(* This function block implements basic functionality for Isolation Gate Valves*)
(* This function block interlock is as follows:
1. The valve can be opened when the difference between the pressures on both sides is
less than the maximum differential pressure.
2. This rule persists until the pressures on both sides are lower than the vacuum-setpoint.
3. Once at-vac, the valve will close if the pressure on either side rises above the setpoint.*)
(*This function block also implements PMPS and EPS interlocks, as well as Fast MPS trigger*)
{attribute 'no_check'}
{attribute 'reflection'} 
FUNCTION_BLOCK FB_VGC_tst Extends FB_Valve
VAR_IN_OUT
	
END_VAR
VAR_INPUT
	(*Upstream Gauge, usually ion gauge*)
	i_stUSG	:	ST_VG;
	(*Downstream Gauge, usually ion gauge*)
	i_stDSG	:	ST_VG;
	{attribute 'pytmc' := '
    pv: Dis_DPIlk
	'}
	i_xDis_DPIlk : BOOL := FALSE;  (* Set to true when calling the function to disable the differential pressure interlock *)
	i_xPMPS_OK:	BOOL	; (*Set to True To switch of the bptm*)
	{attribute 'pytmc' := '
    pv: EPS_OK
	'}
	i_xEPS_OK:	BOOL	:= TRUE; (*External EPS interlock, Set to TRUE when no EPS interlock is required, otherwise set to correct interlock signal*)
	i_xExt_OK: BOOL; (*Other External Interlock, Set to True when no external interlock is required. If this Valve is neigboring a Fast Shutter this should be linked to the fast shutter xVAC_FAULT_OK*)
	i_xOverrideMode : BOOL; (*To be linked to global override bit. This Overrides Vacuum logic only, EPS, MPS and PMPS are still enforces*)
	// Reset fault
	{attribute 'pytmc' := '
    pv: FF_Reset
	'}
    i_xReset: BOOL;
	i_xIsAperture:BOOL :=FALSE; // Set tp True if this is an Aperture Valve, the MPS Fault will trip only when moving.
	i_sDevName : T_MaxString :=  'VGC'; // Device name for diagnostic
	i_nTransitionRootID: UDINT; //A unique transition Root ID that is equal to or greater than 1000
END_VAR
VAR_OUTPUT
	{attribute 'pytmc' := '
    pv:
	'}
	iq_stValve : ST_VGC; (* All valve data and states will be in this struct*)
	
	{attribute 'pytmc' := '
    pv: MPS_FAULT_OK
	field: ZNAM MPS FAULT ;
	field: ONAM MPS OK ;
	'}
	xMPS_OK:	BOOL; (*MPS Fast OK, is set when the Valve is Open*)
END_VAR
VAR_IN_OUT
	io_fbFFHWO    :    FB_HardwareFFOutput;
	fbArbiter: FB_Arbiter();
END_VAR
VAR
	// PMPS
	{attribute 'pytmc' := '
    pv: MPS_OK
	'}
	xPMPS_OK:	BOOL	; (*PMPS interlock*)
	bMoving : BOOL;
	bDone :BOOL;
	tBPTMtimeout:TON;
	 i_nRequestedAssertionID:DWORD;
	bptm: BeamParameterTransitionManager;  
	FFO    :    FB_FastFault :=(
        i_DevName := 'VGC',
        i_Desc := 'Fault occurs when the valve is not in open state',
        i_TypeCode := 16#1010);
	//g_FastFaultOutput1	:	FB_HardwareFFOutput;	

	{attribute 'instance-path'}
	{attribute 'noinit'}
	sPath: STRING;
	
	rDiffPressAllowed	:	REAL := 22.5; // Torr, Default value comes from Vat Valve Manual
	rDiffPress : REAL;
	set : BOOL;
    reset: BOOL;
	  
	xFirstPass	:	BOOL;
	fbFSInit		:	R_TRIG;
	
	tonDelOK : TON;
	rtOK	:	R_TRIG;
	tonOvrd	:	TON;
	rtOpen	:	R_TRIG;
	ftClose: F_TRIG;
	
	tDelOK	:	TIME := T#60S;
	tOvrd	:	TIME := T#10s;
	
	
	(* Timeouts*)
	tTimeOutDuration: TIME:= T#30S;
	tOPNtimeout: TON;
	tCLStimeout:TON;
	
	
	(*IO*)
	i_xOpnLS	AT%I*: BOOL;
	i_xClsLS	AT%I*: BOOL;
	q_xOPN_DO	AT%Q*: BOOL;
    
    // For logging
    eVGCPrevState : E_VGC;
 
	
END_VAR

(* Vacuum gate valve
A. Wallace
16-10-29

A gate valve isolates vacuum volumes. Ideally it can be opened when a system is vented
to allow for faster pumping, and will close when high vacuum is lost.

The following behavior is good for valves in something like a gas attenuator.
This function block does the following:
1. The valve can be opened when the difference between the pressures on both sides is
less than the maximum differential pressure.
2. This rule persists until the pressures on both sides are lower than the vacuum-setpoint.
3. Once at-vac, the valve will close if the pressure on either side rises above the setpoint.

Alternatively, the differential pressure interlock can be disabled so the valve may only be opened
if the pressure on both sides is lower than the at-vacuum-setpoint. You want this behavior if 
the valve is to be used in a UHV section.

Hysteresis is employed to ensure a smooth transition from vented/pumping down, to at-vac.

Finally, an override system is built in so you can bypass all the interlocking logic and 
get back online.
*)
(* 10/1/2018 Margaret Ghaly included EPS, PMPS Checkes and MPS trigger signals*)


fbFSInit( CLK := TRUE, Q => xFirstPass);
(*IO Mapping*)
ACT_IO();

(* On first PLC pass, put valve into vented state, which implies a closed valve *)
IF xFirstPass THEN
	iq_stValve.eVGC_State := Vented;
	iq_stValve.pv_xOPN_SW := FALSE;
	FFO.i_DevName := i_sDevName;
END_IF


///Check valve position
IF iq_stValve.i_xClsLS AND  iq_stValve.i_xOpnLS THEN
	iq_stValve.eState:=INVALID;
ELSIF NOT iq_stValve.i_xClsLS AND iq_stValve.i_xOpnLS AND iq_stValve.q_xOPN_DO THEN 
	iq_stValve.eState:=OPEN;
ELSIF NOT iq_stValve.i_xClsLS AND iq_stValve.i_xOpnLS AND NOT iq_stValve.q_xOPN_DO THEN 
	iq_stValve.eState:=OPEN_F;
ELSIF iq_stValve.i_xClsLS AND NOT iq_stValve.i_xOpnLS AND NOT iq_stValve.q_xOPN_DO THEN 
	iq_stValve.eState:=CLOSED;
ELSIF NOT iq_stValve.i_xClsLS AND NOT iq_stValve.i_xOpnLS THEN 
	iq_stValve.eState:=MOVING;
ELSE
	iq_stValve.eState:=INVALID;
END_IF

// Update hysteresis
///////////////////////////////////////////////////
IF iq_stValve.rAT_VAC_SP_LAST <> iq_stValve.rAT_VAC_SP OR xFirstPass THEN
	iq_stValve.rAT_VAC_SP_LAST := iq_stValve.rAT_VAC_SP;
	iq_stValve.rAT_VAC_HYS := iq_stValve.rHYST_PERC * iq_stValve.rAT_VAC_SP;
END_IF

iq_stValve.rAT_VAC_HYS := LIMIT(0, iq_stValve.rAT_VAC_HYS, iq_stValve.rAT_VAC_SP);
IF iq_stValve.rAT_VAC_SP <> 0 THEN
	IF iq_stValve.rHYST_PERC <> (iq_stValve.rAT_VAC_HYS / iq_stValve.rAT_VAC_SP) THEN
		iq_stValve.rHYST_PERC := LIMIT(0, (iq_stValve.rAT_VAC_HYS / iq_stValve.rAT_VAC_SP) ,1);
	END_IF
END_IF
// Valve at vacuum check
///////////////////////////////////////////////////
	set := i_stUSG.rPRESS < iq_stValve.rAT_VAC_HYS AND i_stDSG.rPRESS < iq_stValve.rAT_VAC_HYS AND i_stUSG.xPRESS_OK AND i_stDSG.xPRESS_OK;
 	iq_stValve.xAT_VAC S= set;
	reset := i_stUSG.rPRESS > iq_stValve.rAT_VAC_SP OR i_stDSG.rPRESS > iq_stValve.rAT_VAC_SP OR NOT i_stUSG.xPRESS_OK OR NOT i_stDSG.xPRESS_OK;
	iq_stValve.xAT_VAC R= reset;
	
// Differential pressure check
///////////////////////////////////////////////////
	(* Calc the differential pressure across the valve *)
	rDiffPress := ABS(i_stUSG.rPRESS - i_stDSG.rPRESS);
	
	(* As long as the differential pressure is less than 30mbar, the valve is allowed to open *)
	IF rDiffPress <= rDiffPressAllowed AND i_stUSG.xPRESS_OK AND i_stDSG.xPRESS_OK THEN
		iq_stValve.xDP_OK := TRUE;
	ELSE
		iq_stValve.xDP_OK	:= FALSE;
		(* If the differential pressure is exceeded, even when the valve is open,
		the state is unexpected and triggers a fault, because it suggests that something
		is wrong with the valve, or gauges or mapping or there is a major leak on one side.*)
		iq_stValve.eVGC_State := ERR_DiffPress;
        iq_stValve.xERR_DifPres := TRUE;
	END_IF

// Valve state
///////////////////////////////////////////////////
CASE iq_stValve.eVGC_State OF
	Vented: (* The Vented state is used during pump down *)        
		(* Assuming the pump down went well, we are now at vacuum on both sides,
		so we move to the vacuum state, otherwise remain in the vented state *)
		IF iq_stValve.xAT_VAC AND (NOT (iq_stValve.xERR_DifPres)) AND (NOT (iq_stValve.xERR_SP)) AND (NOT (iq_stValve.xERR_ExtFault))THEN
		    iq_stValve.eVGC_State := AtVacuum;
		ELSE
		    iq_stValve.eVGC_State := Vented;
		END_IF
	
	AtVacuum:
		IF iq_stValve.xAT_VAC THEN
		(* If both pressure setpoints are made,
		then enable the differential pressure interlock, regardless of the valve state
		assuming we're using some kind of ion gauge where a pressure setpoint cannot be higher than 1E-4 T *)
		iq_stValve.eVGC_State := AtVacuum;
				
		ELSE
		
			(* If the valve is open (or in an unknown state) and either gauge is not at it's vacuum setpoint,
			we have a loss of vacuum error *)
			IF (iq_stValve.i_xOpnLS OR (NOT iq_stValve.i_xOpnLS AND NOT iq_stValve.i_xClsLS)) THEN
				iq_stValve.eVGC_State := ERR_LostVac;
				iq_stValve.xERR_SP := TRUE; //TAW changed this to the ERR_SP bool because I think that's what it was intended to be?
		
			(* Alternatively, if the valve is already closed and we lose pressure on one side,
			it was probably intentional venting, so we calmly move back to venting mode, and
			disable the differential pressure interlock *) //?? 
			ELSIF iq_stValve.i_xClsLS THEN
				iq_stValve.eVGC_State := Vented;
			END_IF
		
		END_IF
	
	ERR_DiffPress:       
		IF NOT (iq_stValve.xERR_DifPres) THEN
			IF iq_stValve.xAT_VAC AND (NOT (iq_stValve.xERR_DifPres)) AND (NOT (iq_stValve.xERR_SP)) AND (NOT (iq_stValve.xERR_ExtFault))THEN
		    	iq_stValve.eVGC_State := AtVacuum;
			ELSE
		    	iq_stValve.eVGC_State := Vented;
			END_IF
		END_IF
		
	
	ERR_LostVac:
		IF NOT (iq_stValve.xERR_SP) THEN
			IF iq_stValve.xAT_VAC AND (NOT (iq_stValve.xERR_DifPres)) AND (NOT (iq_stValve.xERR_SP)) AND (NOT (iq_stValve.xERR_ExtFault))THEN
		    	iq_stValve.eVGC_State := AtVacuum;
			ELSE
		    	iq_stValve.eVGC_State := Vented;
			END_IF
		END_IF
		
	ERR_ExtFault:
		IF NOT (iq_stValve.xERR_ExtFault) AND (i_xExt_OK) THEN
			IF iq_stValve.xAT_VAC AND (NOT (iq_stValve.xERR_DifPres)) AND (NOT (iq_stValve.xERR_SP)) AND (NOT (iq_stValve.xERR_ExtFault))THEN
		    	iq_stValve.eVGC_State := AtVacuum;
			ELSE
		    	iq_stValve.eVGC_State := Vented;
			END_IF
		END_IF
END_CASE

IF (NOT i_xExt_OK) AND (iq_stValve.eState=OPEN)  THEN
	iq_stValve.eVGC_State := ERR_ExtFault;
	iq_stValve.xERR_ExtFault := TRUE;
END_IF

// Interlock evaluation - with bypass for DP ILK bypass
///////////////////////////////////////////////
IF i_xDis_DPIlk THEN
	iq_stValve.xOPN_OK := iq_stValve.xEXT_OK; // AND iq_stValve.xDP_OK ;
ELSE
	iq_stValve.xOPN_OK := iq_stValve.xEXT_OK AND iq_stValve.xAT_VAC;
END_IF


(* Valve operation *)

(* Override logic *)
(* Goal: give ability to override, but do so in a way that people won't forget it.
Solution: Override only after ten seconds of override, protect against blips,
when the valve permission goes true for more than ten seconds consistently, remove override
*)

tonDelOK(IN:=iq_stValve.xOPN_OK, PT:=tDelOK);
rtOK(CLK:=tonDelOK.Q);
IF rtOK.Q AND iq_stValve.pv_xOvrdOpn THEN 
	iq_stValve.pv_xOvrdOpn :=FALSE;
	if (iq_stValve.eState = OPEN) AND (i_xOverrideMode) THEN iq_stValve.pv_xOPN_SW := TRUE; END_IF //for seamless transition   
    //Log
    fbLogger(sMsg:='Override expired', eSevr:=TcEventSeverity.Warning);
END_IF
// Release the Force Open bit when the system override is false
IF NOT (i_xOverrideMode) THEN  iq_stValve.pv_xOvrdOpn :=FALSE; END_IF
//Override timer
tonOvrd(IN:=iq_stValve.pv_xOvrdOpn, PT:=tOvrd);


(* Valve operation *)
(* Here's where we evaluate sw actions and operate the valve *)
(* Valve operation *)

ftClose(CLK:= iq_stValve.pv_xOPN_SW);
rtOpen(CLK:= iq_stValve.pv_xOPN_SW);

(*PMPS OPERATION AND BPTM*)
(*PMPS*)
IF NOT(i_xPMPS_OK) THEN
	ACT_PMPS();
END_IF
xPMPS_OK := i_xPMPS_OK OR (bptm.q_xTransitionAuthorized OR tBPTMtimeout.Q);
(*when interlock is lost the Valve closes regardless of the status of the PMPS and EPS*)
IF NOT (iq_stValve.xOPN_OK) THEN
	iq_stValve.pv_xOPN_SW:= FALSE; // Reset switch after inlk is lost
	iq_stValve.q_xOPN_DO := (iq_stValve.pv_xOPN_SW  AND iq_stValve.xOPN_OK) OR (tonOvrd.Q AND i_xOverrideMode);
ELSIF xPMPS_OK THEN 
	iq_stValve.q_xOPN_DO := (iq_stValve.pv_xOPN_SW  AND iq_stValve.xOPN_OK) OR (tonOvrd.Q AND i_xOverrideMode);
END_IF

(*MPS Fault setting*)
If (i_xIsAperture ) THEN 
	(* When the valve  is open or in Closed position MPS is OK, Fault while moving*)
	xMPS_OK := i_xOpnLS XOR i_xClsLS; 
ELSE
	(* When the valve  is open MPS is OK*)
	xMPS_OK := i_xOpnLS AND NOT i_xClsLS AND q_xOPN_DO; 
END_IF


///Check valve moving postion timout
IF NOT iq_stValve.i_xClsLS AND tCLStimeout.Q THEN 
	iq_stValve.bErrorPresent := TRUE;
	iq_stValve.sErrorMessage := 'Close Timeout';
ELSIF NOT iq_stValve.i_xOpnLS AND tOPNtimeout.Q THEN 
	iq_stValve.bErrorPresent := TRUE; 
	iq_stValve.sErrorMessage := 'Open Timeout';
END_IF
IF (iq_stValve.eState=INVALID) THEN
	iq_stValve.bErrorPresent := TRUE; 
	iq_stValve.sErrorMessage := CONCAT(sPath,'Invalid Valve Position');
END_IF


(*Timers*)
tOPNtimeout(IN:= iq_stValve.q_xOPN_DO, PT := tTimeOutDuration );
tCLStimeout(IN:= NOT iq_stValve.q_xOPN_DO, PT := tTimeOutDuration);


// Alarm reset
//////////////////////////////////////
ACT_ResetAlarms();

(*IO Mapping*)
ACT_IO();

// Log States and triggers
ACT_Logger();



(*FAST FAULT*)
FFO(i_xOK := xMPS_OK,
    i_xReset := i_xReset,
	i_xAutoReset :=TRUE,
    io_fbFFHWO := io_fbFFHWO);

ACTION ACT_IO:
(*inputs*)
iq_stValve.i_xOpnLS := 	i_xOpnLS;
iq_stValve.i_xClsLS:=	i_xClsLS;
iq_stValve.xEXT_OK := i_xEXT_OK;
iq_stValve.xOverrideMode := i_xOverrideMode;
(*outputs*)
q_xOPN_DO:= iq_stValve.q_xOPN_DO;

(*ILK Devices*)
iq_stValve.sIlkUSDeviceName := This^.i_stUSG.sPath;
iq_stValve.sIlkDSDeviceName := This^.i_stDSG.sPath;
END_ACTION

ACTION ACT_Logger:
// ILK logger

IF NOT (iq_stValve.xOPN_OK) AND (ePrevState = OPEN) AND NOT (TonOvrd.Q) THEN
 		fbLogger(sMsg:='Lost interlock ok bit while valve was open.', eSevr:=TcEventSeverity.Critical);  	
END_IF


//Positiong STATE Logger  
IF ePrevState <> iq_stValve.eState THEN
	  CASE iq_stValve.eState OF
		INVALID:
			fbLogger(sMsg:='Valve invalid position.', eSevr:=TcEventSeverity.Critical);
  		MOVING:
			fbLogger(sMsg:='Valve moving', eSevr:=TcEventSeverity.Warning);
		OPEN:
			fbLogger(sMsg:='Valve Open.', eSevr:=TcEventSeverity.Info);
		OPEN_F:
			fbLogger(sMsg:='Valve Open.', eSevr:=TcEventSeverity.Info);
		CLOSED:
			fbLogger(sMsg:='Valve closed.', eSevr:=TcEventSeverity.Info);
	  END_CASE
	  ePrevState := iq_stValve.eState;  
  END_IF
 
 //Pressure STATE Logger  
IF eVGCPrevState <> iq_stValve.eVGC_State THEN
	  CASE iq_stValve.eVGC_State OF
		Vented:
			 fbLogger(sMsg:='Vented', eSevr:=TcEventSeverity.Info);
  		AtVacuum:
			 fbLogger(sMsg:='Vacuum setpoint satisfied', eSevr:=TcEventSeverity.Info);
		ERR_DiffPress:
			 fbLogger(sMsg:='Potential accidental vent.', eSevr:=TcEventSeverity.Critical);
		ERR_LostVac:
			fbLogger(sMsg:='Unexpected loss of vacuum while valve was open or moving.', eSevr:=TcEventSeverity.Critical);
		ERR_ExtFault:
			 fbLogger(sMsg:='Lost external interlock while valve was open.', eSevr:=TcEventSeverity.Critical);
	  END_CASE
	  eVGCPrevState := iq_stValve.eVGC_State;  
  END_IF
  


// Log valve timeouts
tErrorPresent(CLK:=iq_stValve.bErrorPresent);
IF tErrorPresent.Q THEN fbLogger(sMsg:=iq_stValve.sErrorMessage, eSevr:=TcEventSeverity.Warning); END_IF

// Log valve open
tAction(CLK:= iq_stValve.q_xOPN_DO);
IF tAction.Q THEN fbLogger(sMsg:='Valve commanded open', eSevr:=TcEventSeverity.Info); END_IF

// Log override mode enabled
tOverrideActivated(CLK:= (tonOvrd.Q AND i_xOverrideMode));
IF tOverrideActivated.Q THEN fbLogger(sMsg:='Valve override mode activated', eSevr:=TcEventSeverity.Warning); END_IF
END_ACTION

ACTION ACT_PMPS:
bMoving := (iq_stValve.pv_xOPN_SW AND iq_stValve.i_xClsLS) XOR (NOT iq_stValve.pv_xOPN_SW AND i_xOpnLS);
bDone := (iq_stValve.pv_xOPN_SW AND iq_stValve.i_xOpnLS) XOR (NOT iq_stValve.pv_xOPN_SW AND i_xClsLS);
If (i_xIsAperture ) OR (iq_stValve.pv_xOPN_SW )THEN
	bptm.i_stRequestedAssertion := PMPS_GVL.cstFullBeam;
ELSE  bptm.i_stRequestedAssertion := PMPS_GVL.cstSafeBeam;
END_IF

bptm(fbArbiter:=fbArbiter,
     i_TransitionAssertionID:=i_nTransitionRootID+2,
     i_stTransitionAssertion:=PMPS_GVL.cstSafeBeam,
     i_nRequestedAssertionID:=i_nTransitionRootID+ BOOL_TO_UDINT( iq_stValve.pv_xOPN_SW),
     i_stRequestedAssertion:=,
     i_xMoving:=,//bMoving,
     i_xDoneMoving:= bDone,
     stCurrentBeamParameters:=PMPS_GVL.stCurrentBeamParameters,
     q_xTransitionAuthorized=>);
// Timeout
tBPTMtimeout(IN:= bMoving AND NOT bptm.q_xTransitionAuthorized, PT:=T#2S);
//xPMPS_OK := bptm.q_xTransitionAuthorized OR tBPTMtimeout.Q;
//xPMPS_OK := i_xPMPS_OK OR (bptm.q_xTransitionAuthorized OR tBPTMtimeout.Q); // Moved to FB, move it back after testing

//Timeout and clear request
IF (tBPTMtimeout.Q) THEN
	fbArbiter.RemoveRequest(bptm.i_TransitionAssertionID);
	fbArbiter.RemoveRequest(bptm.i_nRequestedAssertionID);
END_IF
END_ACTION

ACTION ACT_ResetAlarms:
iq_stValve.xERR_DifPres R= iq_stValve.pv_xAlmRst;
iq_stValve.xERR_SP R= iq_stValve.pv_xAlmRst;
iq_stValve.bErrorPresent R= iq_stValve.pv_xAlmRst;
iq_stValve.xERR_ExtFault R= iq_stValve.pv_xAlmRst;

IF ( iq_stValve.pv_xAlmRst) THEN
	iq_stValve.sErrorMessage :='';
	 iq_stValve.pv_xAlmRst := FALSE;
END_IF
END_ACTION

METHOD PUBLIC M_IsClosed : BOOL
VAR_INPUT
END_VAR
M_IsClosed := (This^.iq_stValve.eState = E_ValvePositionState.CLOSED);
END_METHOD

METHOD PUBLIC M_IsOpen : BOOL
VAR_INPUT
END_VAR
M_IsOpen := (This^.iq_stValve.eState = E_ValvePositionState.OPEN);
END_METHOD

// Use this Methode to Open or close the valve by setting the OPN_SW to the input value.
METHOD PUBLIC M_Set_OPN_SW : BOOL
VAR_INPUT
		value:BOOL;
END_VAR
This^.iq_stValve.pv_xOPN_SW := value;
END_METHOD

END_FUNCTION_BLOCK

(* stored: Version 1.1.0.1, ProductVersion 3.1.4024.3
   POU FB_VGC_tst: Id {c11ab03e-606b-4cce-9b4d-159d1fcd34a6}, SpecialFunc None
   Action ACT_IO: Id {49200a75-822d-4181-a7dc-7357ab320676}
   Action ACT_Logger: Id {33c734b4-18eb-497c-97c5-1c03caae0a85}
   Action ACT_PMPS: Id {681d3417-9168-4ed2-a720-6960ced65f1e}
   Action ACT_ResetAlarms: Id {9a7577da-26b2-495c-9589-68c6c7e48602}
   Method M_IsClosed: Id {7adfcd87-1ead-47b1-8d3b-7ff8725e8bf2}
   Method M_IsOpen: Id {926d4a16-d991-4fd9-8eeb-248145693117}
   Method M_Set_OPN_SW: Id {2bb21d3e-078f-41ea-a609-e838be4e8d88} *)
